// TIA Portal V17 export
// export: Created 2023-03-08T16:44:23.1874801Z, ExportSetting None, DisplayName Totally Integrated Automation Portal, DisplayVersion V17 Update 4, DisplayName TIA Portal Openness, DisplayVersion V17 Update 4, DisplayName TIA Portal Version Control Interface, DisplayVersion V17, DisplayName STEP 7 Professional, DisplayVersion V17 Update 4, DisplayName STEP 7 Safety, DisplayVersion V17, DisplayName WinCC Advanced / Unified PC, DisplayVersion V17 Update 4
DATA_BLOCK "DI"   // DB12
{ S7_Optimized_Access := 'TRUE' }
// stored: AutoNumber false, MemoryReserve 100
   VAR
      ZSC_33303 : Bool;   // SOV EBV 33303 CLOSE FEEDBACK
      ZSO_33303 : Bool;   // SOV EBV 33303 OPEN FEEDBACK
      ZSC_33304 : Bool;   // SOV EBV 33304 CLOSE FEEDBACK
      ZSO_33304 : Bool;   // SOV EBV 33304 OPEN FEEDBACK
      ZSC_33305 : Bool;   // SOV EBV 33305 CLOSE FEEDBACK
      ZSO_33305 : Bool;   // SOV EBV 33305 OPEN FEEDBACK
      TSH_33304A : Bool;   // HEATER A TEMPERATURE
      TSH_33304B : Bool;   // HEATER B TEMPERATURE
      TSH_33304C : Bool;   // HEATER C TEMPERATURE
      TSH_33304D : Bool;   // HEATER D TEMPERATURE
      ZSC_33302 : Bool;   // SOV ABV 33302 CLOSE FEEDBACK
      ZSO_33302 : Bool;   // SOV ABV 33302 OPEN FEEDBACK
      XS_33302 : Bool;   // COMPRESSOR MAIN MOTOR RUNNING FEEDBACK
      XF_33302 : Bool;   // COMPRESSOR MAIN MOTOR FAULT FEEDBACK
      XS_33329A : Bool;   // LUBE OIL PUMP M341A RUNNING FEEDBACK
      XF_33328A : Bool;   // LUBE OIL PUMP M341A FAULT FEEDBACK
      XS_33329B : Bool;   // LUBE OIL PUMP M341B RUNNING FEEDBACK
      XF_33328B : Bool;   // LUBE OIL PUMP M341B FAULT FEEDBACK
      XY_33324A : Bool;   // HEATER A RUNNING FEEDBACK
      XF_33320 : Bool;   // HEATER A FAULT FEEDBACK
      XY_33324B : Bool;   // HEATER B RUNNING FEEDBACK
      XF_33321 : Bool;   // HEATER B FAULT FEEDBACK
      XY_33324C : Bool;   // HEATER C RUNNING FEEDBACK
      XF_33322 : Bool;   // HEATER C FAULT FEEDBACK
      XY_33324D : Bool;   // HEATER D RUNNING FEEDBACK
      XF_33323 : Bool;   // HEATER D FAULT FEEDBACK
      HS_33301A : Bool;   // START UNIT
      HS_33302A : Bool;   // STOP UNIT
      HS_33304A : Bool;   // RESET
      HS_33307 : Bool;   // UNIT MAINTENANCE
      EY_33332 : Bool;   // PERMISSION TO START FROM DCS
      EY_33311 : Bool;   // TRIP FROM DCS
      HS_33399 : Bool;   // EMERGENCY PB ON LCP-333-01
      TSH_33399 : Bool;   // LCP-333-01 INTERNAL HIGH TEMPERATURE
      XA_33399 : Bool;   // LCP-333-01 24VDC POWER SUPPLY MALFUNCTION
      LSHH_33306 : Bool;   // ECONOMIZER LEVEL SWITCH
      LSHH_33308 : Bool;   // KO DRUM LEVEL SWITCH
   END_VAR
BEGIN
END_DATA_BLOCK
